Yaskawa INFORM job: SYS_VERIFY_GATE_LOCKED.JBI

/JOB
//NAME SYS_VERIFY_GATE_LOCKED
//POS
///NPOS 0,0,0,0,0,0
//INST
///DATE 2022/07/18 11:55
///ATTR SC,RW
///GROUP1 RB1
NOP
WAIT IN#(1)=OFF
END
